// Core §8.9 — apply the one generated priority/category to a diagnostic at its
// source. Unknown external reasons keep the caller values until their owning
// AlarmLog joins a validated runtime record.
FUNCTION F_RationalizeDiagnostic : BOOL
VAR_IN_OUT
    Diag : ST_Diagnostic;
END_VAR
VAR
    meta : ST_AlarmMeta;
END_VAR

F_RationalizeDiagnostic := F_ReasonMeta(
    Reason := Diag.ReasonCode, Meta := meta);
IF F_RationalizeDiagnostic THEN
    Diag.Severity := meta.Priority;
    Diag.Category := meta.Category;
END_IF

END_FUNCTION

(* stored: Version 1.1.0.1, ProductVersion 3.1.4024.12
   POU F_RationalizeDiagnostic: Id {cb0e4b63-f458-42d7-a908-ae706e4639c2}, SpecialFunc None *)
